PROGRAM MAIN
VAR
	
ACS380 		: ABB_ACS380;

xReady 		: BOOL;
xRun 		: BOOL;
xStop 		: BOOL;
xEstop		: BOOL;
xReset		: BOOL;
xJog		: BOOL;
xFaultPresent : BOOL;
iSpeedRef 	: INT;

END_VAR

//Need to be True
ACS380.ControlWord.REMOTE_CMD := TRUE;
ACS380.ControlWord.RAMP_OUT_ZERO := TRUE;
ACS380.ControlWord.RAMP_HOLD := TRUE;
ACS380.ControlWord.RAMP_IN_ZERO := TRUE;

//VFD Reset
	IF xReset THEN
		ACS380.ControlWord.RESET := TRUE;
	ELSE
		ACS380.ControlWord.RESET := FALSE;
	END_IF

//Stop Not Active
	IF NOT xStop AND NOT xEstop  THEN
		ACS380.ControlWord.OFF2_CONTROL := TRUE;
		ACS380.ControlWord.OFF3_CONTROL := TRUE;
	ELSE
		ACS380.ControlWord.OFF2_CONTROL := FALSE;
		ACS380.ControlWord.OFF3_CONTROL := FALSE;
	END_IF
	
//VFD Ready
	IF xReady AND ACS380.StatusWord.RDY_ON AND NOT ACS380.StatusWord.TRIPPED AND NOT xFaultPresent THEN
		ACS380.ControlWord.OFF1_CONTROL := TRUE;
	ELSE
		ACS380.ControlWord.OFF1_CONTROL := FALSE;
	END_IF
	
//Run VFD
	IF xRun AND ACS380.StatusWord.RDY_RUN THEN
		ACS380.ControlWord.RUN := TRUE;
	ELSE
		ACS380.ControlWord.RUN := FALSE;
	END_IF

//VFD Speed Command
	ACS380.SpeedCMD := iSpeedRef;
	
//VFD Fault
	IF ACS380.StatusWord.TRIPPED OR ACS380.ComError THEN
		xFaultPresent := TRUE;
	ELSIF xFaultPresent AND xReset THEN
		xFaultPresent := FALSE;
	END_IF

END_PROGRAM

(* stored: Version 1.1.0.1, ProductVersion 3.1.4024.12
   POU MAIN: Id {65ddfae7-441d-40a9-83f4-805b218a5035}, SpecialFunc None *)
